// TIA Portal V16 export
// export: Created 2023-03-29T11:05:04.8999597Z, ExportSetting WithDefaults, DisplayName Totally Integrated Automation Portal, DisplayVersion V16 Update 6, DisplayName TIA Portal Version Control Interface, DisplayVersion V16 Update 2, DisplayName TIA Portal Openness, DisplayVersion V16 Update 6, DisplayName STEP 7 Professional, DisplayVersion V16 Update 6, DisplayName STEP 7 Safety, DisplayVersion V16, DisplayName WinCC Advanced, DisplayVersion V16 Update 6
VAR_GLOBAL   // PLC tag table "Z11"
   isReadyZ11 AT %M85.3 : Bool;
   inputAwariaMomentZ11 AT %M85.4 : Bool;
   inputOtwartaZ11 AT %M85.5 : Bool;
   inputZamkniętaZ11 AT %M85.6 : Bool;
   inputRuchZ11 AT %M85.7 : Bool;
   setSVMO_Z11 AT %M13.6 : Bool;   // Znacznik polecenia otwórz w trybie automat
   inputmodeAutZ11 AT %M17.6 : Bool;   // Znacznik trybu pracy 1=Aut, 0=Rem
   inputAumalokalneZ11 AT %M87.2 : Bool;
   inputAumaautomatZ11 AT %M87.3 : Bool;
   inputAumagotowośćZ11 AT %M87.4 : Bool;
   inputAumaawariaZ11 AT %M87.5 : Bool;
   setSVMC_Z11 AT %M13.7 : Bool;   // Znacznik polecenia zamknij w trybie automat
   CMD_Open_Z11 AT %M33.3 : Bool;   // załącz otwieranie Z11
   CMD_Close_Z11 AT %M33.4 : Bool;   // załącz zamykanie Z11
   CMD_Awaria_Z11 AT %M91.2 : Bool;   // Awaria zbiorcza
   setAlarm_Moment_Z11 AT %M91.3 : Bool;   // znacznik alarmu od momentówki w trybie zdalnym (aut/mamnual)
   bitH_Alarm_Z11 AT %M95.0 : Bool;   // Alarm - kopia sygału z instancji DB10
   bitH_Open_Z11 AT %M95.1 : Bool;   // Otwarta - kopia sygału z instancji DB10
   bitH_REM_Z11 AT %M95.2 : Bool;   // Zdalne - kopia sygału z instancji DB10
   bitH_Close_Z11 AT %M95.3 : Bool;   // Zamknięta - kopia sygału z instancji DB10
   bitH_Opening_Z11 AT %M95.4 : Bool;   // sygnał otwórz- kopia sygału z instancji DB10
   bitH_Res_Z11 AT %M95.6 : Bool;   // sygnał reset - kopia sygału z instancji DB10
   bitH_Aut_Man_Z11 AT %M95.7 : Bool;   // sygnał aut=1, manual =0 - kopia sygału z instancji DB10
   bitH_Closing_Z11 AT %M95.5 : Bool;   // sygnał zamknij- kopia sygału z instancji DB10
   Byte_Status_Z11 AT %MB95 : Byte;   // status napędu
END_VAR
